FUNCTION_BLOCK FB_Base
VAR_OUTPUT
    nCnt : INT;
END_VAR

METHOD METH_DoAlso : BOOL
VAR_INPUT
END_VAR
METH_DoAlso := TRUE;
END_METHOD

METHOD METH_DoIt : BOOL
nCnt := -1;
END_METHOD

END_FUNCTION_BLOCK

(* stored: Version 1.1.0.1, ProductVersion 3.1.4024.12
   POU FB_Base: Id {04bdcdb3-c29d-42e9-a8c0-67506a1767dd}, SpecialFunc None
   Method METH_DoAlso: Id {486720d1-1192-44f3-a26e-44a4f7d6874b}
   Method METH_DoIt: Id {df5c08b4-7e27-4c2d-afc5-50a98e6eee76} *)
